Staubli VAL3: onF3Event.pgx

program onF3Event()
  local num i
  local num l_nSize[3]
  local num l_nType
  local string l_sProg
  local string l_sFill
  local num j
begin
  // look if the bButton is enable
  if bButton[2]
    // generate the file of the production
    call processList:makeFile()
  endIf
end
